{attribute 'no_assign'}
FUNCTION_BLOCK FB_Mover IMPLEMENTS I_Mover
VAR_INPUT
END_VAR
VAR_OUTPUT
END_VAR
VAR
	_bIsInitialized: BOOL;	

	fbPlanarMover : MC_PlanarMover;
	fbPlanarFeedback: MC_PlanarFeedback;
	trackTrail: MC_PlanarTrackTrail;
	SyncMoverFeedback: Tc3_Mc3PlanarMotion.MC_PlanarFeedbackGearInPosOnTrackWithMasterMover;
	
	_GearInOptions: Tc3_Mc3PlanarMotion.ST_GearInPosOnTrackWithMasterMoverOptions;
	_stMoveOnTrackOptions: ST_MoveOnTrackOptions;
	_stLeaveSystemAtOptions : ST_LeaveSystemAtOptions;
	
	_syncTrail : MC_PlanarTrackTrail;
	
	CmdFeedback :  XtsCommandFeedback;
	ipXtsMover:   I_XtsXlMover1;
	ipXtsProcessingUnit:  I_XtsProcessingUnit1;

	_stMoverInfos : ST_MoverInfo;	
	_stMoverOnTrackInfos : MC_MOVER_ON_TRACK_INFORMATION;

	_nextMcTrackOid: OTCID;
	_stDynamics: DynamicConstraint_PathXY;
	_TargetTrack : UDINT;
	_ReWork : BOOL;
	_partConfig: UINT;
	_InSync :BOOL; 
	_PositionOnTrack : LREAL;
	_Track : OTCID; 
	_distToEndOfTrack : LREAL;

	fbResult						: FB_TcMessage;
///	_ipComObject					: ITComObject;
	PID_OnTrackInfos				: PTCID := 16#05030180;
	bInit 							: BOOL;
	nErrorID						: HRESULT; 
	ControllerOID					: otcid;
	stPointerAddresses				: ST_PointerAddresses;
	ScopeVariables					: ST_ScopeValues;
	
END_VAR

METHOD ClearSyncTrail : BOOL
VAR_INPUT
END_VAR
_syncTrail.Clear();

IF _syncTrail.TrackCount = 0 THEN
	ClearSyncTrail := TRUE;
END_IF
END_METHOD



METHOD CycleUpdate : BOOL


VAR_INST
	_trackEnum: e_TrackNum;

END_VAR
IF NOT _bIsInitialized THEN
	RETURN;
END_IF

fbPlanarMover.GetTrackTrailInformation(trackTrail);
_PositionOnTrack := fbPlanarMover.MCTOPLC.SETONTRACK.SetPos;


fbPlanarMover.Update();
fbPlanarFeedback.Update();
SyncMoverFeedback.Update();
UpdateXtsTrack();
GetOnTrackInfos(fbPlanarMover.MCTOPLC.STD.MoverOID) ;


_stMoverinfos.MoverOtcid :=fbPlanarMover.MCTOPLC.STD.MoverOID ;
_stMoverinfos.IsActive := ipXtsMover.GetIsActive(0);
_stMoverinfos.ActPos :=  ipXtsMover.GetPositionInfo_trackPosition(0);
_stMoverinfos.ActVelo := fbPlanarMover.MCTOPLC.SETONTRACK.SetVelo;
_stMoverinfos.IsVirtuell := ipXtsMover.GetIsVirtualFeedbackEnabled(0);
_stMoverinfos.Positition :=	fbPlanarMover.MCTOPLC.SETONTRACK.SetPos;
_stMoverinfos.Track := TO_STRING(_trackEnum);
_stMoverinfos.Error := fbPlanarMover.Error;
_stMoverinfos.ErrorID := fbPlanarMover.ErrorId;
_stMoverinfos.PlanarMoverCommandMode :=  TO_STRING(fbPlanarMover.MCTOPLC.STD.CommandMode);
_stMoverinfos.State :=  TO_STRING(fbPlanarMover.MCTOPLC.STD.State);
_stMoverinfos.Gap := _stMoverOnTrackInfos.Gap;
_stMoverinfos.LimitAcc := _stMoverOnTrackInfos.Limits.A;
_stMoverinfos.LimitDec := _stMoverOnTrackInfos.Limits.D;
_stMoverinfos.LimitJerk := _stMoverOnTrackInfos.Limits.J;
_stMoverinfos.LimitVelo := _stMoverOnTrackInfos.Limits.V;
_stMoverinfos.TargetTrackPosition := _stMoverOnTrackInfos.TargetPosition.Position;
_stMoverinfos.TargetTrack := _stMoverOnTrackInfos.TargetPosition.TrackOid;
_stMoverinfos.RemainingDistance := _stMoverOnTrackInfos.Remainingdistance;
ScopeVariables.ActStatus := ipXtsMover.GetDriveStatus(0);
IF stPointerAddresses.ActHwPosModuloPointer <> 0 THEN
	ScopeVariables.ActHwPosModulo := stPointerAddresses.ActHwPosModuloPointer^ ;
	ScopeVariables.ActPosError := stPointerAddresses.ActPosErrorPointer^ ;
	ScopeVariables.ActVelo := stPointerAddresses.ActVeloPointer^ ;
	ScopeVariables.SetAccItp := stPointerAddresses.SetAccItpPointer^;
	ScopeVariables.SetCurrent := stPointerAddresses.SetCurrentPointer^ ;
	ScopeVariables.SetVeloItp := stPointerAddresses.SetVeloItpPointer^  ;
	ScopeVariables.SetForce := stPointerAddresses.SetForcePointer^;

END_IF
END_METHOD

METHOD Disable : BOOL
VAR_INPUT
END_VAR
fbPlanarMover.Enable(
	commandFeedback:= fbPlanarFeedback);
	
Disable :=fbPlanarFeedback.Done OR fbPlanarFeedback.Error;
END_METHOD

METHOD Enable : BOOL
VAR_INPUT
END_VAR
fbPlanarMover.Disable(
	commandFeedback:= fbPlanarFeedback);
	
Enable :=fbPlanarFeedback.Done OR fbPlanarFeedback.Error;
END_METHOD

METHOD GetActHwPosModuloPointer : POINTER TO LREAL
VAR_INPUT
	ControllerOID : OTCID;
END_VAR
VAR
	ipComObject			: ITcWatchSource;
	oidActHwPosModulo	: OTCID := 16#A0000010;
	sizeData			: UDINT;
	adrData 			: PVOID; 
END_VAR

nErrorID := FW_ObjMgr_GetObjectInstance(	oid		:=	ControllerOID, 
											iid		:=	TC_GLOBAL_IID_LIST.IID_ITcWatchSource, 
											pipUnk 	:= ADR(ipComObject));


																				
IF ipComObject <> 0 THEN
	
	sizeData := SIZEOF(GetActHwPosModuloPointer);
	adrData := ADR(GetActHwPosModuloPointer);

	nErrorID := ipComObject.InterpretGroupOffsetLength( 	indexOffset := oidActHwPosModulo ,
															cbLength 	:= sizeData,
															ppData 		:= adrData);
	ipComObject.TcRelease();	
	ipComObject := 0;													
														
												
END_IF
END_METHOD

METHOD GetActPosErrorPointer : POINTER TO LREAL
VAR_INPUT
	ControllerOID : OTCID;
END_VAR
VAR
	ipComObject			: ITcWatchSource;
	oidActPosError		: OTCID := 16#A0000018;
	sizeData			: UDINT;
	adrData 			: PVOID; 
END_VAR

nErrorID := FW_ObjMgr_GetObjectInstance(	oid		:=	ControllerOID, 
											iid		:=	TC_GLOBAL_IID_LIST.IID_ITcWatchSource, 
											pipUnk 	:= ADR(ipComObject));


																				
IF ipComObject <> 0 THEN
	
	sizeData := SIZEOF(GetActPosErrorPointer);
	adrData := ADR(GetActPosErrorPointer);

	nErrorID := ipComObject.InterpretGroupOffsetLength( 	indexOffset := oidActPosError ,
															cbLength 	:= sizeData,
															ppData 		:= adrData);
	ipComObject.TcRelease();	
	ipComObject := 0;													
														
												
END_IF
END_METHOD

METHOD GetActVeloPointer : POINTER TO LREAL
VAR_INPUT
	ControllerOID : OTCID;
END_VAR
VAR
	ipComObject			: ITcWatchSource;
	oidActVelo	: OTCID := 16#A0000008;
	sizeData			: UDINT;
	adrData 			: PVOID; 
END_VAR

nErrorID := FW_ObjMgr_GetObjectInstance(	oid		:=	ControllerOID, 
											iid		:=	TC_GLOBAL_IID_LIST.IID_ITcWatchSource, 
											pipUnk 	:= ADR(ipComObject));


																				
IF ipComObject <> 0 THEN
	
	sizeData := SIZEOF(GetActVeloPointer);
	adrData := ADR(GetActVeloPointer);

	nErrorID := ipComObject.InterpretGroupOffsetLength( 	indexOffset := oidActVelo ,
															cbLength 	:= sizeData,
															ppData 		:= adrData);
	ipComObject.TcRelease();	
	ipComObject := 0;													
														
												
END_IF
END_METHOD

METHOD GetDistanceToEot : LREAL
VAR_INPUT
	TrackLenght : LREAL;
END_VAR
GetDistanceToEot := _distToEndOfTrack;

IF fbPlanarMover.MCTOPLC.SETONTRACK.TrackOID<>0 THEN 
	GetDistanceToEot := TrackLenght-fbPlanarMover.MCTOPLC.SETONTRACK.SetPos;
END_IF
END_METHOD

METHOD GetOnTrackInfos : BOOL
VAR_INPUT
	nObjectId : otcid; 
END_VAR
VAR
	nData 			: UDINT := SIZEOF(_stMoverOnTrackInfos);
	pData 			: PVOID := ADR(_stMoverOnTrackInfos);
	stEventEntry	: TcEventEntry;
	pstEventEntry	: REFERENCE TO TcEventEntry REF= stEventEntry;
END_VAR
VAR_INST
	hResult : HRESULT;
	bError : BOOL;
	_ipComObject : ITComObject;
END_VAR
bError := FALSE;


IF nObjectId <> 0 AND_THEN _ipComObject = 0 THEN
	 FW_ObjMgr_GetObjectInstance(	oid		:= nObjectId, 
								iid		:= TC_GLOBAL_IID_LIST.IID_ITComObject, 
								pipUnk	:= ADR(_ipComObject)) ;
END_IF

IF _ipComObject <> 0 THEN 
	 hResult := 	_ipComObject.TcgetObjPara(		pid := PID_OnTrackInfos,
													nData := nData,
													pData := pData,
													pgp := 0); 	
	IF hResult = 0 THEN
		GetOnTrackInfos := TRUE;
ELSE
	HRESULTAdsErr_TO_TcEventEntry(hResult,stEventEntry);
	IF NOT fbResult.EqualsToEventEntryEx( stOther := stEventEntry) THEN
		fbResult.CreateEx(stEventEntry, 0);
		fbResult.Send(0);
		fbResult.Release();
	END_IF
		bError := TRUE;
	END_IF							
END_IF
END_METHOD

METHOD GetSetAccItpPointer : POINTER TO LREAL
VAR_INPUT
	ControllerOID : OTCID;
END_VAR
VAR
	ipComObject			: ITcWatchSource;
	oidSetAccItp		: OTCID := 16#A0000038;
	sizeData			: UDINT;
	adrData 			: PVOID; 
END_VAR

nErrorID := FW_ObjMgr_GetObjectInstance(	oid		:=	ControllerOID, 
											iid		:=	TC_GLOBAL_IID_LIST.IID_ITcWatchSource, 
											pipUnk 	:= ADR(ipComObject));


																				
IF ipComObject <> 0 THEN
	
	sizeData := SIZEOF(GetSetAccItpPointer);
	adrData := ADR(GetSetAccItpPointer);

	nErrorID := ipComObject.InterpretGroupOffsetLength( 	indexOffset := oidSetAccItp ,
															cbLength 	:= sizeData,
															ppData 		:= adrData);
	ipComObject.TcRelease();	
	ipComObject := 0;													
														
												
END_IF
END_METHOD

METHOD GetSetCurrentPointer : POINTER TO LREAL
VAR_INPUT
	ControllerOID : OTCID;
END_VAR
VAR
	ipComObject			: ITcWatchSource;
	oidSetCurrent 		: OTCID := 16#A0000048;
	sizeData			: UDINT;
	adrData 			: PVOID; 
END_VAR

nErrorID := FW_ObjMgr_GetObjectInstance(	oid		:=	ControllerOID, 
											iid		:=	TC_GLOBAL_IID_LIST.IID_ITcWatchSource, 
											pipUnk 	:= ADR(ipComObject));


																				
IF ipComObject <> 0 THEN
	
	sizeData := SIZEOF(GetSetCurrentPointer);
	adrData := ADR(GetSetCurrentPointer);

	nErrorID := ipComObject.InterpretGroupOffsetLength( 	indexOffset := oidSetCurrent ,
															cbLength 	:= sizeData,
															ppData 		:= adrData);
	ipComObject.TcRelease();	
	ipComObject := 0;													
														
												
END_IF
END_METHOD

METHOD GetSetForcePointer : POINTER TO LREAL
VAR_INPUT
	ControllerOID : OTCID;
END_VAR
VAR
	ipComObject			: ITcWatchSource;
	oidSetForce 		: OTCID := 16#A0000050;
	sizeData			: UDINT;
	adrData 			: PVOID; 
END_VAR

nErrorID := FW_ObjMgr_GetObjectInstance(	oid		:=	ControllerOID, 
											iid		:=	TC_GLOBAL_IID_LIST.IID_ITcWatchSource, 
											pipUnk 	:= ADR(ipComObject));


																				
IF ipComObject <> 0 THEN
	
	sizeData := SIZEOF(GetSetForcePointer);
	adrData := ADR(GetSetForcePointer);

	nErrorID := ipComObject.InterpretGroupOffsetLength( 	indexOffset := oidSetForce ,
															cbLength 	:= sizeData,
															ppData 		:= adrData);
	ipComObject.TcRelease();	
	ipComObject := 0;													
														
												
END_IF
END_METHOD

METHOD GetSetVeloItpPointer : POINTER TO LREAL
VAR_INPUT
	ControllerOID : OTCID;
END_VAR
VAR
	ipComObject			: ITcWatchSource;
	oidSetVeloItp	: OTCID := 16#A0000030;
	sizeData			: UDINT;
	adrData 			: PVOID; 
END_VAR

nErrorID := FW_ObjMgr_GetObjectInstance(	oid		:=	ControllerOID, 
											iid		:=	TC_GLOBAL_IID_LIST.IID_ITcWatchSource, 
											pipUnk 	:= ADR(ipComObject));


																				
IF ipComObject <> 0 THEN
	
	sizeData := SIZEOF(GetSetVeloItpPointer);
	adrData := ADR(GetSetVeloItpPointer);

	nErrorID := ipComObject.InterpretGroupOffsetLength( 	indexOffset := oidSetVeloItp ,
															cbLength 	:= sizeData,
															ppData 		:= adrData);
	ipComObject.TcRelease();	
	ipComObject := 0;													
														
												
END_IF
END_METHOD

METHOD Halt : BOOL
VAR_INPUT
END_VAR
fbPlanarMover.Halt(
	commandFeedback:= fbPlanarFeedback, 
	constraint:= _stDynamics);
	
Halt :=fbPlanarFeedback.Done OR fbPlanarFeedback.Error;
END_METHOD

METHOD Init : BOOL
VAR_INPUT

	XtsMover:   I_XtsXlMover1;
	XtsProcessingUnit :  I_XtsProcessingUnit1;

	
END_VAR
VAR_STAT
	Getpointer : BOOL;
END_VAR


ipXtsMover:= XtsMover;
ipXtsProcessingUnit :=  XtsProcessingUnit;




ControllerOID:= ipXtsMover.GetMoverController(CmdFeedback);
IF ControllerOID <> 0  THEN
	stPointerAddresses.ActHwPosModuloPointer := GetActHwPosModuloPointer(ControllerOID);
	stPointerAddresses.SetVeloItpPointer := GetSetVeloItpPointer(ControllerOID);
	stPointerAddresses.ActVeloPointer := GetActVeloPointer(ControllerOID);
	stPointerAddresses.SetAccItpPointer := GetSetAccItpPointer(ControllerOID);
	stPointerAddresses.ActPosErrorPointer := GetActPosErrorPointer(ControllerOID);
	stPointerAddresses.SetCurrentPointer := GetSetCurrentPointer(ControllerOID); 
	stPointerAddresses.SetForcePointer := GetSetForcePointer(ControllerOID); 
	bInit:=TRUE;
	
	
END_IF
			
IF    CmdFeedback.IsDone THEN
	_bIsInitialized := TRUE;
	Init := TRUE;
END_IF
END_METHOD

METHOD JoinNearestTrack : BOOL
VAR_INPUT 
	aMcTracks : ARRAY[*] OF MC_PlanarTrack;
	Trackcount : UINT;
END_VAR

VAR_INST
	nForCounter: UINT;
	mcTrackOid: OTCID;
	partOid: OTCID;
	cmdFeedback					: 	XtsCommandFeedback;
	objectInfo: PlanarObjectInfo;
END_VAR
partOid := ipXtsMover.GetPositionInfo_partObjectId(cmdFeedback);

IF partOid = 0 THEN
	RETURN;
END_IF

IF cmdFeedback.IsDone THEN
	mcTrackOid := ipXtsProcessingUnit.XlPartWithOid(partOid, cmdFeedback).GetMcTrackOid(cmdFeedback);
	
	FOR nForCounter := 1 TO Trackcount DO
		objectInfo := aMcTracks[nForCounter].GetPlanarObjectInfo();
		IF objectInfo.Id = mcTrackOid THEN
			fbPlanarMover.JoinTrack(fbPlanarFeedback, aMcTracks[nForCounter], _stDynamics, 0); 
			RETURN;
		END_IF
	END_FOR
END_IF
END_METHOD

METHOD LeaveSystemAt : BOOL
VAR_INPUT
	ConnectionOut: REFERENCE TO MC_PlanarTrackConnectionOut;
	gap : LREAL; 
END_VAR
_stLeaveSystemAtOptions.gap := gap;
_stLeaveSystemAtOptions.gapMode := MC_GAP_MODE_ON_TRACK.Fast1D; 
_stLeaveSystemAtOptions.dynamicMode :=  MC_DYNAMIC_MODE_ON_TRACK.None;

fbPlanarMover.LeaveSystemAt(fbPlanarFeedback, ConnectionOut,  _stDynamics,_stLeaveSystemAtOptions);
END_METHOD

METHOD MoveOnTrack : BOOL
VAR_INPUT
	track: REFERENCE TO MC_PlanarTrack;	
	targetPos: LREAL;
	gap : LREAL; 
END_VAR
_stMoveonTrackOptions.gap := gap; 

fbPlanarMover.MoveOnTrack(
	commandFeedback:= fbPlanarFeedback, 
	targetTrack:= track, 
	targetPositionOnTrack:= targetPos, 
	constraint:= _stDynamics, 
	options:= _stMoveOnTrackOptions);
END_METHOD

PROPERTY MoverStopped : BOOL
GET
MoverStopped := (fbPlanarMover.MCTOPLC.SETONTRACK.SetVelo < 20);
END_GET
SET
END_SET
END_PROPERTY

PROPERTY P_Dynamics : REFERENCE TO DynamicConstraint_PathXY;
GET

P_Dynamics REF= _stDynamics;
END_GET
END_PROPERTY

PROPERTY P_IsInitialized : bool
GET
P_IsInitialized := _bIsInitialized;
END_GET
END_PROPERTY

PROPERTY P_MoveOnTrackOptions  : REFERENCE TO  ST_MoveOnTrackOptions
GET
P_MoveOnTrackOptions REF= _stMoveOnTrackOptions;
END_GET
END_PROPERTY

PROPERTY P_MoverInfos : REFERENCE TO ST_MoverInfo
GET
P_MoverInfos  REF= _stMoverInfos;
END_GET
END_PROPERTY

PROPERTY p_MoverOTCID : OTCID
GET
p_MoverOTCID := fbPlanarMover.MCTOPLC.STD.MoverOID;
END_GET
SET
END_SET
END_PROPERTY

PROPERTY P_PlanarFeedback : REFERENCE TO MC_PlanarFeedback
GET
P_PlanarFeedback REF= fbPlanarFeedback;
END_GET
END_PROPERTY

PROPERTY P_PlanarMover :   REFERENCE TO  MC_PlanarMover
GET
P_PlanarMover REF= fbPlanarMover;
END_GET
END_PROPERTY

PROPERTY P_ScopeVariables  :   REFERENCE TO ST_ScopeValues
GET
 P_ScopeVariables   REF= ScopeVariables;
END_GET
END_PROPERTY

PROPERTY P_SyncFeedback :  REFERENCE TO MC_PlanarFeedbackGearInPosOnTrackWithMasterMover
GET
P_SyncFeedback REF= SyncMoverFeedback;
END_GET
END_PROPERTY

PROPERTY P_TargetTrack : UDINT
GET
P_TargetTrack := _TargetTrack ;
END_GET
SET
_TargetTrack := P_TargetTrack;
END_SET
END_PROPERTY

PROPERTY Rework : BOOL
GET
Rework := _Rework;
END_GET
SET
_Rework := Rework;
END_SET
END_PROPERTY

METHOD SetSyncTrail : BOOL
VAR_INPUT
	PlanarTrack : MC_PlanarTrack;
END_VAR
_syncTrail.AddTrack(track:= PlanarTrack);///GVL_Mc.aMCTracks[E_TrackNum.Small]); 
 
SetSyncTrail := TRUE;
END_METHOD

METHOD SyncToOtherMover : BOOL
VAR_INPUT
	masterSyncPos : LREAL; // Position on the master track
	followerSyncPos : LREAL; // position on the follower track
	PlanarMoverToFollow: REFERENCE TO Tc3_Mc3PlanarMotion.MC_PlanarMover;
	masterTrack : REFERENCE TO Tc3_Mc3PlanarMotion.MC_PlanarTrack; 
	followerTrack : REFERENCE TO Tc3_Mc3PlanarMotion.MC_PlanarTrack; 
	velo : REFERENCE TO LREAL; 
END_VAR

VAR
	trail: Tc3_Mc3PlanarMotion.MC_PlanarTrackTrail;

END_VAR
_GearInOptions.allowedSlaveSyncDirections := MC_SYNC_DIRECTIONS.Positive; 
_GearInOptions.directionMasterSyncPosition := MC_DIRECTION.mcDirectionNonModulo; 
_GearInOptions.directionSlaveSyncPosition := MC_DIRECTION.mcDirectionNonModulo;  
_GearInOptions.followMover := FALSE; 
_GearInOptions.gap := 0; // elimnate gap funciton 
_GearInOptions.inSyncToleranceDistance :=0; 
_GearInOptions.moduloToleranceMasterSyncPosition := 0; 
_GearInOptions.moduloToleranceSlaveSyncPosition := 0;  
_stDynamics.V := velo; 

fbPlanarMover.GearInPosOnTrackWithMasterMover(
	commandFeedback:=  SyncMoverFeedback , 
	masterMover:= PlanarMoverToFollow , 
	trackTrail:= _syncTrail, // may need to give a trail maybe not
	masterSyncPosition:= masterSyncPos, 
	masterSyncPositionTrack:= MasterTrack , 
	slaveSyncPosition:= followerSyncPos, 
	slaveSyncPositionTrack:= followerTrack, 
	constraint:=_stDynamics , 
	options:=_GearInOptions );
END_METHOD

METHOD PUBLIC UpdateXtsTrack
VAR_INPUT
END_VAR
VAR_STAT
	nTrackCount: UINT;
	oid1: OTCID;
	oid2: OTCID;
	
	nForCounter: UINT;
	nPartConfigCount: UINT;
	
	partConfig1: OTCID;
	partConfig2: OTCID;
	
	mcTrackOid1: OTCID;
	mcTrackOid2: OTCID;
	trackOid: OTCID;
	
	nTrackTrailCount: UDINT;
	actTrackOid: OTCID;
	nIndexInTrail: UDINT;
END_VAR
nTrackTrailCount := trackTrail.TrackCount;
actTrackOid := fbPlanarMover.MCTOPLC.SETONTRACK.TrackOID;

IF nTrackTrailCount <= 1 THEN
	RETURN;
END_IF

FOR nForCounter := 1 TO UDINT_TO_UINT(nTrackTrailCount) DO
	oid1 := trackTrail.GetTrackOidAt(nForCounter);
	IF oid1 = actTrackOid THEN
		IF nForCounter < nTrackTrailCount THEN
			oid2 := trackTrail.GetTrackOidAt(nForCounter + 1);
			EXIT;
		ELSE
			RETURN; //last one ine track trail
		END_IF
	END_IF
END_FOR

IF oid2 = _nextMcTrackOid AND ipXtsMover.GetPositionInfo_partPosition(CmdFeedback) < 600 THEN //no change
	RETURN;
END_IF

nTrackCount := ipXtsProcessingUnit.TrackCount();

FOR nForCounter := 1 TO nTrackCount DO
	nPartConfigCount := ipXtsProcessingUnit.Track(nForCounter, CmdFeedback).PartConfigCount(); 
	
	IF nPartConfigCount >= 2  THEN
		partConfig1 := ipXtsProcessingUnit.Track(nForCounter, CmdFeedback).GetPartConfigOidAt(1, 0);
		partConfig2 := ipXtsProcessingUnit.Track(nForCounter, CmdFeedback).GetPartConfigOidAt(2, 0);
//
		
		IF partConfig1 = 0 OR partConfig2 = 0 THEN
			CONTINUE;
		END_IF
		
		mcTrackOid1 := ipXtsProcessingUnit.XlPartWithOid(partConfig1, CmdFeedback).GetMcTrackOid(0);
		mcTrackOid2 := ipXtsProcessingUnit.XlPartWithOid(partConfig2, CmdFeedback).GetMcTrackOid(0);
		IF mcTrackOid1 = oid1 AND mcTrackOid2 = oid2   THEN
			trackOid := ipXtsProcessingUnit.Track(nForCounter, CmdFeedback).GetObjectId();
			ipXtsMover.SetActiveTrackObjectId(trackOid, CmdFeedback);
			
			IF CmdFeedback.IsDone THEN
				_nextMcTrackOid := oid2;
			END_IF
			
			RETURN;
		END_IF
	END_IF
END_FOR
END_METHOD

PROPERTY XlProcessingUnit : I_XtsProcessingUnit1
GET
XlProcessingUnit := ipXtsProcessingUnit;
END_GET
END_PROPERTY

PROPERTY XtsComFeed : REFERENCE TO  XtsCommandFeedback
GET
XtsComFeed REF= CmdFeedback;
END_GET
END_PROPERTY

PROPERTY XtsXlMover : I_XtsXlMover1
GET
XtsXlMover := ipXtsMover;
END_GET
END_PROPERTY

END_FUNCTION_BLOCK

(* stored: Version 1.1.0.1
   POU FB_Mover: Id {198fd53d-d7b4-4fcb-b2eb-8f7ae59664d7}, SpecialFunc None
   Folder Methods: Id {0af15190-d2aa-44a0-bb66-f7b3132dbfa1}
   Folder Pointer: Id {88a55610-b4ba-442c-901c-a1d5c38e9c09}
   Folder Properties: Id {7031571e-e1d9-43e7-ab72-63d8e981e89e}
   Method ClearSyncTrail: Id {e61bcda0-90c3-4136-81ce-acf5e5eb8d9e}
   Method CycleUpdate: Id {f03058aa-6296-4ef4-9484-d5b71f801a75}
   Method Disable: Id {d4cd6619-4c4b-49cb-88a3-5d2e4721828c}
   Method Enable: Id {8f81c7e1-1425-40e9-94a8-fc8dd0ad962e}
   Method GetActHwPosModuloPointer: Id {545ee952-faf6-4fbe-a77f-0166a9d43d19}
   Method GetActPosErrorPointer: Id {2ecd72a2-84a2-4a71-957c-596e585b1820}
   Method GetActVeloPointer: Id {585ee1f2-7235-4fbd-8162-a4589b32290e}
   Method GetDistanceToEot: Id {e9f79926-9abd-432b-bf12-313fbb070747}
   Method GetOnTrackInfos: Id {80c76236-e464-41c7-ade3-18309c2f7e10}
   Method GetSetAccItpPointer: Id {38fda956-3272-4366-8ea8-4b26a0282b1a}
   Method GetSetCurrentPointer: Id {32bf2739-ffc9-4f88-809c-ec244e04556a}
   Method GetSetForcePointer: Id {e894f5dd-5b0b-4403-9709-99392ce01d9d}
   Method GetSetVeloItpPointer: Id {e3a179d5-a2c3-4c5b-a620-b5edc38673c5}
   Method Halt: Id {be2a5a02-47df-4fd0-9ccd-24499830f258}
   Method Init: Id {64dda721-646a-4cf1-ab7d-9993c2a9294b}
   Method JoinNearestTrack: Id {7049d311-b9c1-401e-88ee-2d1a43482209}
   Method LeaveSystemAt: Id {6b5686b0-ff62-458e-8370-b6983356eb85}
   Method MoveOnTrack: Id {5cb1162f-8066-466b-a4ab-0b247e872c60}
   Property MoverStopped: Id {04d60936-8878-4099-a93e-51ae708d75d9}
   Get Get: Id {64097993-7eee-4f83-926e-27b475cbba5d}
   Set Set: Id {a44d7ebb-539a-4a0d-bb16-c43cb3963f38}
   Property P_Dynamics: Id {1ecca715-6941-4f72-8708-bfc5f157ffb4}
   Get Get: Id {266d93a2-8578-440a-b579-03e9192f6cab}
   Property P_IsInitialized: Id {b7011b40-0827-4f2c-9967-dcf04f3d6670}
   Get Get: Id {d30e5ad4-0da0-42fb-aa4d-b6ece7f34840}
   Property P_MoveOnTrackOptions: Id {fb69dd5d-5a1c-486a-a084-fed687cabe26}
   Get Get: Id {f3d0f320-9269-4a8e-a547-66ab76d6278d}
   Property P_MoverInfos: Id {e247c7bf-cf6b-4d35-b73d-b6630d38bcfa}
   Get Get: Id {0f87cb2e-58c3-4156-bf2a-d5c34dbd43ec}
   Property p_MoverOTCID: Id {ce0ba360-bc0d-42ad-8903-9adb5e1a2946}
   Get Get: Id {916509e8-dbb2-4754-93e1-b2ed765f430f}
   Set Set: Id {c0f1b337-663c-40ea-8d0e-69d3d272f5d2}
   Property P_PlanarFeedback: Id {21da37fd-6f26-475d-beab-c040fa3e1691}
   Get Get: Id {106a1958-6758-4ec6-83fb-080c48933bcd}
   Property P_PlanarMover: Id {ade24b6b-bd49-4670-bd83-4d8ea4dd5ac9}
   Get Get: Id {caf06972-2707-423e-a74b-61e4467a57c5}
   Property P_ScopeVariables: Id {0e6cd576-6eaf-462d-bdfc-d05925d0a9ea}
   Get Get: Id {a01be95f-411e-4419-b450-aff9fde2de05}
   Property P_SyncFeedback: Id {d85f38ed-ffc5-44d4-bfc1-afe7972a3eda}
   Get Get: Id {7aadb2e2-7225-49aa-b6ad-e4a667efb167}
   Property P_TargetTrack: Id {aa403c76-568e-4bf9-873b-2566a88e0af2}
   Get Get: Id {7a918e8e-93e7-4fae-bb7b-36deca07c1de}
   Set Set: Id {3d2068f3-914a-4c88-8f32-0932e316ce68}
   Property Rework: Id {0e60f93b-c652-4b1d-8202-d7b886cfe370}
   Get Get: Id {b329ade1-87a9-43ab-bcc1-eb939538692d}
   Set Set: Id {94b726a9-11fd-4d67-885a-4ff8be4a2d21}
   Method SetSyncTrail: Id {8774251d-30e6-45ca-a10f-4e71c1952ba8}
   Method SyncToOtherMover: Id {9903c21e-709d-4928-99f6-93578aa23443}
   Method UpdateXtsTrack: Id {21f4b176-5457-4b67-bca0-ab7203ad0675}
   Property XlProcessingUnit: Id {c937fd04-ede7-4a06-bb80-d96e27dc80d2}
   Get Get: Id {6798c177-744f-424d-8da8-6f37f30325e6}
   Property XtsComFeed: Id {77a11faf-2343-4c02-8b32-d650545bd2e9}
   Get Get: Id {7f9d7ec5-c980-4ab6-b02b-3ce27efef18a}
   Property XtsXlMover: Id {70d89129-e56a-44f9-bf01-7348e90e5b05}
   Get Get: Id {211069c9-c1df-40ce-bc0d-73dbdefcb458} *)
